// TIA Portal V20 export
DATA_BLOCK "Config"   // DB116
// stored: MemoryReserve 100, Namespace Unit1.Em12
   VAR
      em : "LAF_typeEmConfiguration";   // Configuration of EM Parameters
      cmStackNgBoxDetect : "LBC_typeDigitalSignalConfiguration";
      cmStackNgBoxFullDetect : "LBC_typeDigitalSignalConfiguration";
      cmStackNgBoxLoadingUpDown : "LBC_typeTwoWayActuatorConfiguration";
      cmStackNgBoxUnitMoverBwdFwd : "LBC_typeTwoWayActuatorConfiguration";
      cmStackNgBoxClampLeftOpenClose : "LBC_typeTwoWayActuatorConfiguration";
      cmStackNgBoxClampRightOpenClose : "LBC_typeTwoWayActuatorConfiguration";
      cmStackNgBoxClampMoverOpenClose : "LBC_typeTwoWayActuatorConfiguration";
      cmStackNgBoxLiftDownUp : "LBC_typeTwoWayActuatorConfiguration";
      cmStackNgBoxLockDownUp : "LBC_typeTwoWayActuatorConfiguration";
   END_VAR
BEGIN
   em.referenceDesignator.parent := WSTRING#'U1';
   em.referenceDesignator.relative := WSTRING#'EM0';
   cmStackNgBoxLoadingUpDown.referenceDesignator := WSTRING#'NG CLAMP Z-Axis';
   cmStackNgBoxLoadingUpDown.monitoringDiscrepancy := T#5s;
   cmStackNgBoxUnitMoverBwdFwd.referenceDesignator := WSTRING#'NG CLAMP UNIT MOVER';
   cmStackNgBoxUnitMoverBwdFwd.monitoringDiscrepancy := T#5s;
   cmStackNgBoxClampLeftOpenClose.referenceDesignator := WSTRING#'NG CLAMP LEFT';
   cmStackNgBoxClampLeftOpenClose.monitoringDiscrepancy := T#5s;
   cmStackNgBoxClampRightOpenClose.referenceDesignator := WSTRING#'NG CLAMP RIGHT';
   cmStackNgBoxClampRightOpenClose.monitoringDiscrepancy := T#5s;
   cmStackNgBoxClampMoverOpenClose.referenceDesignator := WSTRING#'NG CLAMP MOVER';
   cmStackNgBoxClampMoverOpenClose.monitoringDiscrepancy := T#5s;
   cmStackNgBoxLiftDownUp.referenceDesignator := WSTRING#'NG BOX LIFT';
   cmStackNgBoxLiftDownUp.monitoringDiscrepancy := T#5s;
   cmStackNgBoxLockDownUp.referenceDesignator := WSTRING#'NG BOX LOCK';
   cmStackNgBoxLockDownUp.monitoringDiscrepancy := T#5s;
END_DATA_BLOCK
